TYPE ASCF_CC_OPCUACS_ConnectionStatus :
STRUCT
	Status			: DINT		:= 0;
	ServerState		: DINT		:= 0;
	ServiceLevel	: USINT		:= 0;
END_STRUCT
END_TYPE

(* stored: Version 1.1.0.1, ProductVersion 3.1.4026.4
   DUT ASCF_CC_OPCUACS_ConnectionStatus: Id {3a1d2694-6f89-4a8d-b720-1dff697d1902} *)
